# EPICS autosave request: blurApp/Db/NDBlur_settings.req
file "NDPluginBase_settings.req", P=$(P), R=$(R)
$(P)$(R)KernelWidth
$(P)$(R)KernelHeight
$(P)$(R)BlurType
